Staubli VAL3: MotionQueue.dtx

public num nPush
public num nPop
public num nElems
public MotionBuffer buffer[10]
  [0]
    mdesc mVelAcc = {leave=0, reach=0}
    num nDuration
    num nSequence
    jointRx jJointRx
  [1]
    mdesc mVelAcc = {leave=0, reach=0}
    num nDuration
    num nSequence
    jointRx jJointRx
  [2]
    mdesc mVelAcc = {leave=0, reach=0}
    num nDuration
    num nSequence
    jointRx jJointRx
  [3]
    mdesc mVelAcc = {leave=0, reach=0}
    num nDuration
    num nSequence
    jointRx jJointRx
  [4]
    mdesc mVelAcc = {leave=0, reach=0}
    num nDuration
    num nSequence
    jointRx jJointRx
  [5]
    mdesc mVelAcc = {leave=0, reach=0}
    num nDuration
    num nSequence
    jointRx jJointRx
  [6]
    mdesc mVelAcc = {leave=0, reach=0}
    num nDuration
    num nSequence
    jointRx jJointRx
  [7]
    mdesc mVelAcc = {leave=0, reach=0}
    num nDuration
    num nSequence
    jointRx jJointRx
  [8]
    mdesc mVelAcc = {leave=0, reach=0}
    num nDuration
    num nSequence
    jointRx jJointRx
  [9]
    mdesc mVelAcc = {leave=0, reach=0}
    num nDuration
    num nSequence
    jointRx jJointRx
